// TIA Portal V15.1 export
// export: Created 2020-06-12T07:35:47.2880859Z, ExportSetting None, DisplayName Totally Integrated Automation Portal, DisplayVersion V15.1, DisplayName TIA Portal Openness, DisplayVersion V15.1, DisplayName STEP 7 Professional, DisplayVersion V15.1, DisplayName STEP 7 Safety, DisplayVersion V15.1, DisplayName WinCC Advanced, DisplayVersion V15.1
FUNCTION "Gas_ctrl" : Void   // FC2, FBD
TITLE = Gas system
{ S7_Optimized_Access := 'TRUE' }
// This is a simple 1-line systsem which works in the modes:
// * Keep constant pressure (use fixed flow to reach a target pressure)
// * Keep constant flow (use controllable flow to compensate a gas leakages and a dedusting suction)
// * flood the mold and hood by defined gas volume
// stored: SetENOAutomatically False
   VAR_TEMP
      tActFlow : Real;
      tFloodAmount : Real;   // Temp calculation flood gas amount
      tLinePress : Real;
      tSetFlow : Real;
      tActPress : Real;
      _csf : Bool;
      tRun : Bool;   // Pre Flooding active
      tRunForFlooding : Bool;   // Flooding active
      tDoAmount : Bool;
      tStop : Bool;
      tAutoOn : Bool;
      tReqOn : Bool;
      tReqOff : Bool;
      tReqPressOn : Bool;
      tReqPressOff : Bool;
      tReqAmountOn : Bool;
      tReqAmountOff : Bool;
      tAutoOff : Bool;
      tReqAmountReset : Bool;
      tReqDummy : Bool;
      tGasOn : Bool;
      tAutoMode : Int;
      tMeasFlow : Real;
      tDoPressConst : Bool;
      tDoFlowConst : Bool;
      tCurrSetFlow : Real;
      tAutoIsOn : Bool;
      tPressAboveSet : Real;
      tGasBlowOn : Bool;
   END_VAR
   VAR_TEMP   // added for the SCL form of the ladder/FBD networks
      _w1 : Bool;
      _w2 : Bool;
   END_VAR
BEGIN

REGION Network 1: COMMON SYSTEM FAULT
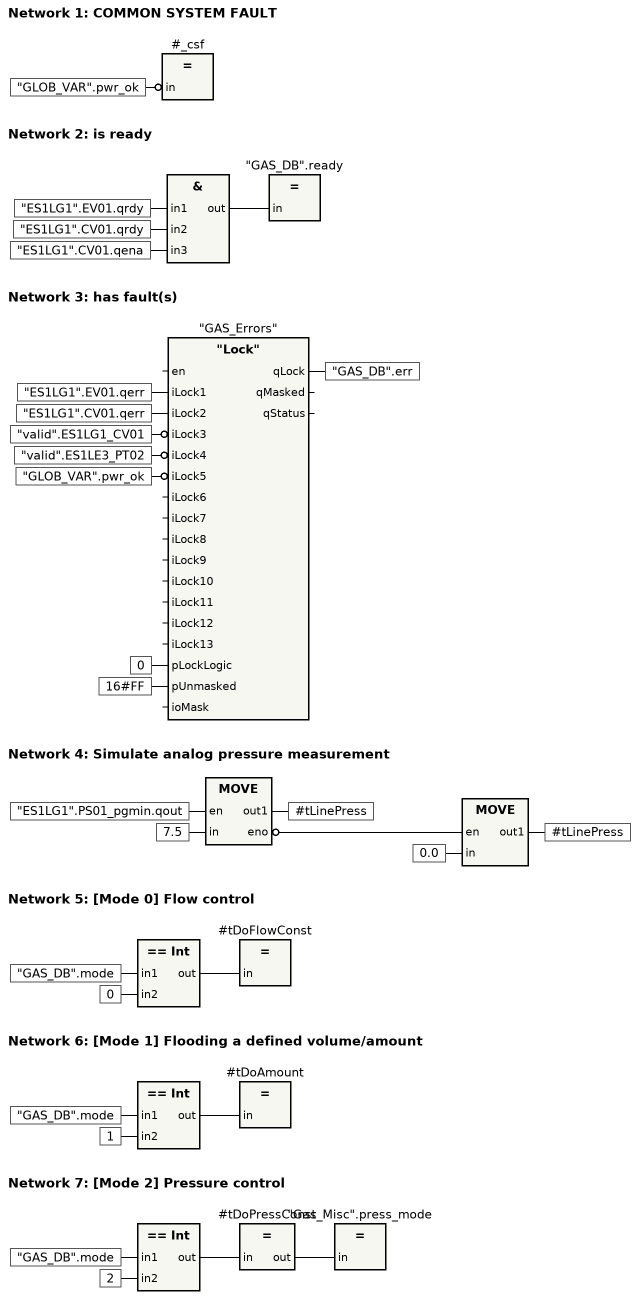
   #_csf := NOT "GLOB_VAR".pwr_ok;
END_REGION

REGION Network 2: is ready
   "GAS_DB".ready := "ES1LG1".EV01.qrdy AND "ES1LG1".CV01.qrdy AND "ES1LG1".CV01.qena;
END_REGION

REGION Network 3: has fault(s)
   "GAS_Errors"(iLock1 := "ES1LG1".EV01.qerr,   // "Lock"
                iLock2 := "ES1LG1".CV01.qerr,
                iLock3 := NOT "valid".ES1LG1_CV01,
                iLock4 := NOT "valid".ES1LE3_PT02,
                iLock5 := NOT "GLOB_VAR".pwr_ok,
                pLockLogic := 0,
                pUnmasked := 16#FF,
                qLock => "GAS_DB".err);
END_REGION

REGION Network 4: Simulate analog pressure measurement
   IF "ES1LG1".PS01_pgmin.qout THEN #tLinePress := 7.5; END_IF;
   IF NOT "ES1LG1".PS01_pgmin.qout THEN #tLinePress := 0.0; END_IF;
END_REGION

REGION Network 5: [Mode 0] Flow control
   #tDoFlowConst := "GAS_DB".mode = 0;
END_REGION

REGION Network 6: [Mode 1] Flooding a defined volume/amount
   #tDoAmount := "GAS_DB".mode = 1;
END_REGION

REGION Network 7: [Mode 2] Pressure control
   #tDoPressConst := "GAS_DB".mode = 2;
   "Gas_Misc".press_mode := #tDoPressConst;
END_REGION

REGION Network 8: Flow set: flow const
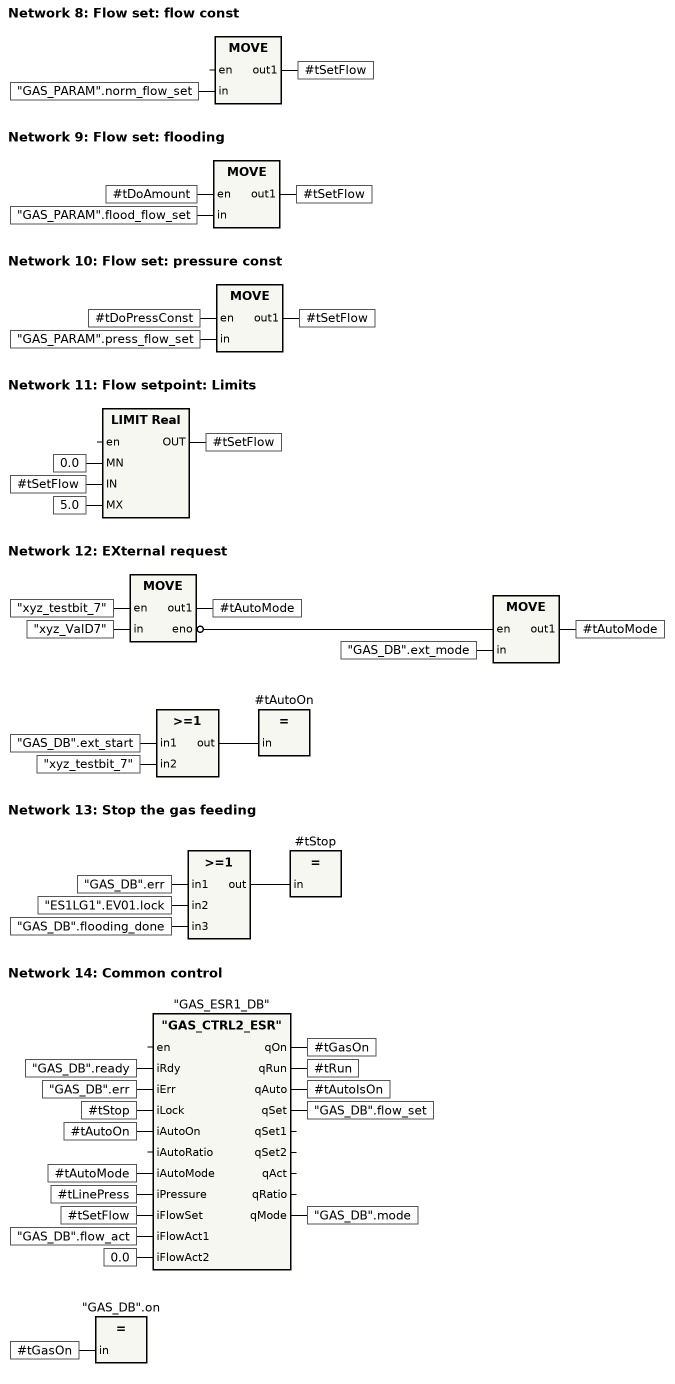
   #tSetFlow := "GAS_PARAM".norm_flow_set;
END_REGION

REGION Network 9: Flow set: flooding
   IF #tDoAmount THEN #tSetFlow := "GAS_PARAM".flood_flow_set; END_IF;
END_REGION

REGION Network 10: Flow set: pressure const
   IF #tDoPressConst THEN #tSetFlow := "GAS_PARAM".press_flow_set; END_IF;
END_REGION

REGION Network 11: Flow setpoint: Limits
   #tSetFlow := LIMIT(MN := 0.0, IN := #tSetFlow, MX := 5.0);
END_REGION

REGION Network 12: EXternal request
   IF "xyz_testbit_7" THEN #tAutoMode := "xyz_ValD7"; END_IF;
   IF NOT "xyz_testbit_7" THEN #tAutoMode := "GAS_DB".ext_mode; END_IF;
   #tAutoOn := "GAS_DB".ext_start OR "xyz_testbit_7";
END_REGION

REGION Network 13: Stop the gas feeding
   #tStop := "GAS_DB".err OR "ES1LG1".EV01.lock OR "GAS_DB".flooding_done;
END_REGION

REGION Network 14: Common control
   "GAS_ESR1_DB"(iRdy := "GAS_DB".ready,   // "GAS_CTRL2_ESR"
                 iErr := "GAS_DB".err,
                 iLock := #tStop,
                 iAutoOn := #tAutoOn,
                 iAutoMode := #tAutoMode,
                 iPressure := #tLinePress,
                 iFlowSet := #tSetFlow,
                 iFlowAct1 := "GAS_DB".flow_act,
                 iFlowAct2 := 0.0,
                 qOn => #tGasOn,
                 qRun => #tRun,
                 qAuto => #tAutoIsOn,
                 qSet => "GAS_DB".flow_set,
                 qMode => "GAS_DB".mode);
   "GAS_DB".on := #tGasOn;
END_REGION

REGION Network 15: M1> Flooding is requested
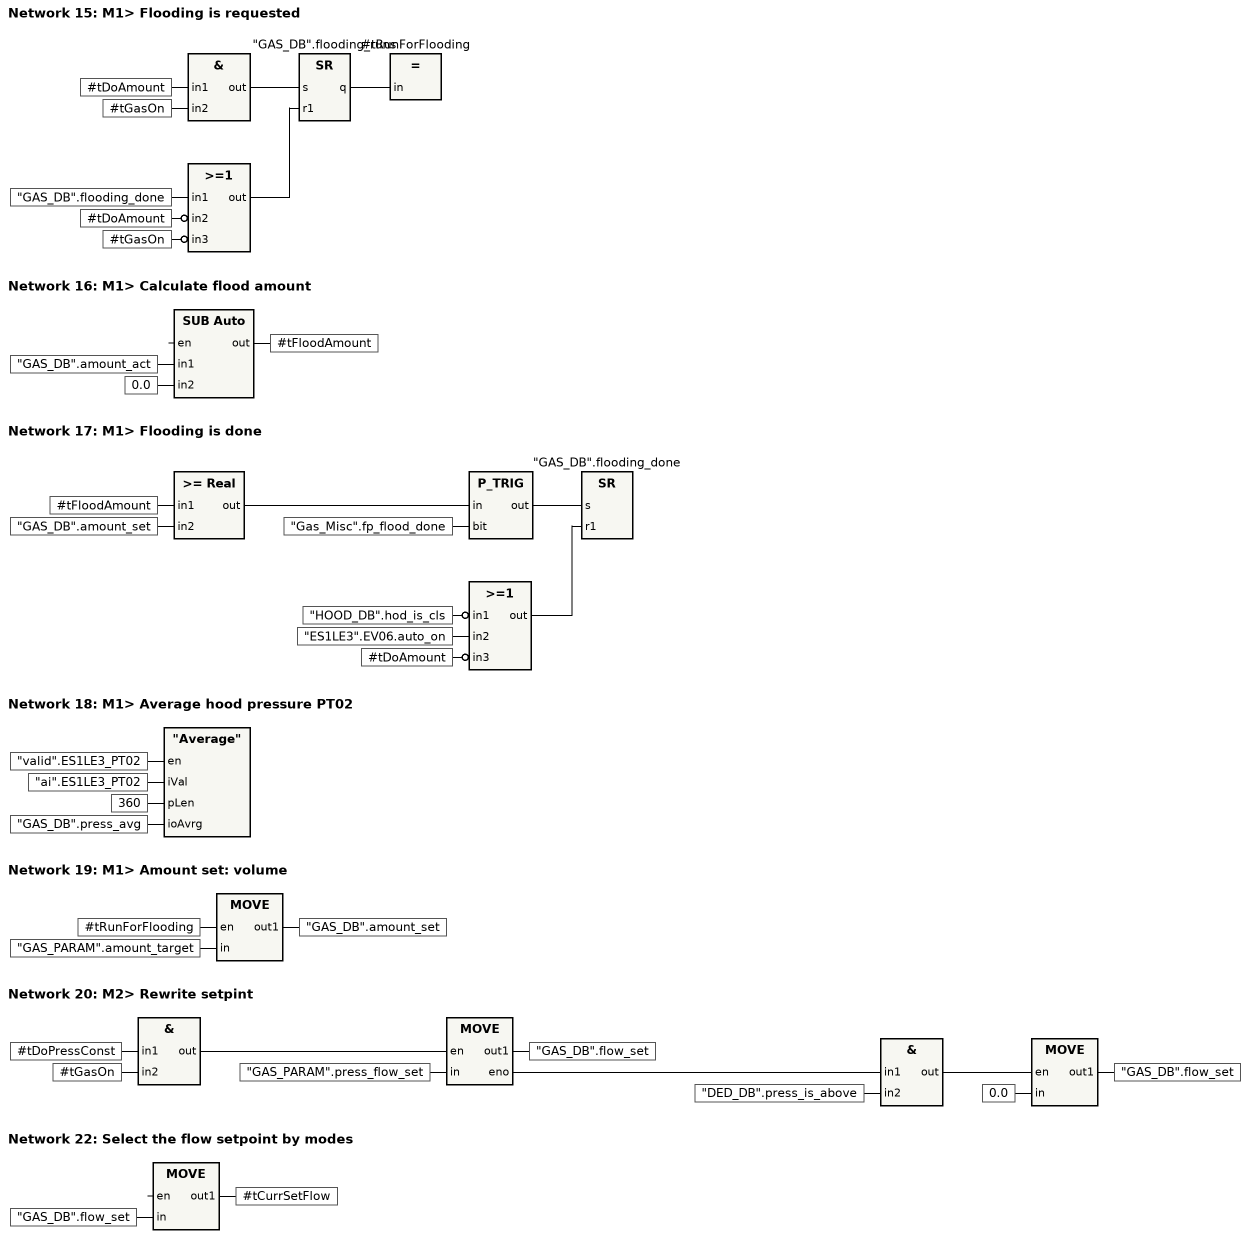
   IF #tDoAmount AND #tGasOn THEN
       "GAS_DB".flooding_runs := TRUE;   // SR flip-flop
   END_IF;
   IF "GAS_DB".flooding_done OR NOT #tDoAmount OR NOT #tGasOn THEN "GAS_DB".flooding_runs := FALSE; END_IF;
   #tRunForFlooding := "GAS_DB".flooding_runs;
END_REGION

REGION Network 16: M1> Calculate flood amount
   #tFloodAmount := "GAS_DB".amount_act - 0.0;
END_REGION

REGION Network 17: M1> Flooding is done
   #_w1 := #tFloodAmount >= "GAS_DB".amount_set;
   #_w2 := #_w1 AND NOT "Gas_Misc".fp_flood_done;   // rising edge
   "Gas_Misc".fp_flood_done := #_w1;
   IF #_w2 THEN
       "GAS_DB".flooding_done := TRUE;   // SR flip-flop
   END_IF;
   IF NOT "HOOD_DB".hod_is_cls OR "ES1LE3".EV06.auto_on OR NOT #tDoAmount THEN
       "GAS_DB".flooding_done := FALSE;
   END_IF;
END_REGION

REGION Network 18: M1> Average hood pressure PT02
   IF "valid".ES1LE3_PT02 THEN
       "Average"(iVal := "ai".ES1LE3_PT02, pLen := 360, ioAvrg := "GAS_DB".press_avg);
   END_IF;
END_REGION

REGION Network 19: M1> Amount set: volume
   IF #tRunForFlooding THEN "GAS_DB".amount_set := "GAS_PARAM".amount_target; END_IF;
END_REGION

REGION Network 20: M2> Rewrite setpint
   // FIXME: this is trick :( It should be re-factored
   #_w1 := #tDoPressConst AND #tGasOn;
   IF #_w1 THEN "GAS_DB".flow_set := "GAS_PARAM".press_flow_set; END_IF;
   IF #_w1 AND "DED_DB".press_is_above THEN "GAS_DB".flow_set := 0.0; END_IF;
END_REGION

REGION Network 21: ******************************
END_REGION

REGION Network 22: Select the flow setpoint by modes
   #tCurrSetFlow := "GAS_DB".flow_set;
END_REGION

REGION Network 23: Actual flow (emulation)
   // THis is using because a measurement is not correct
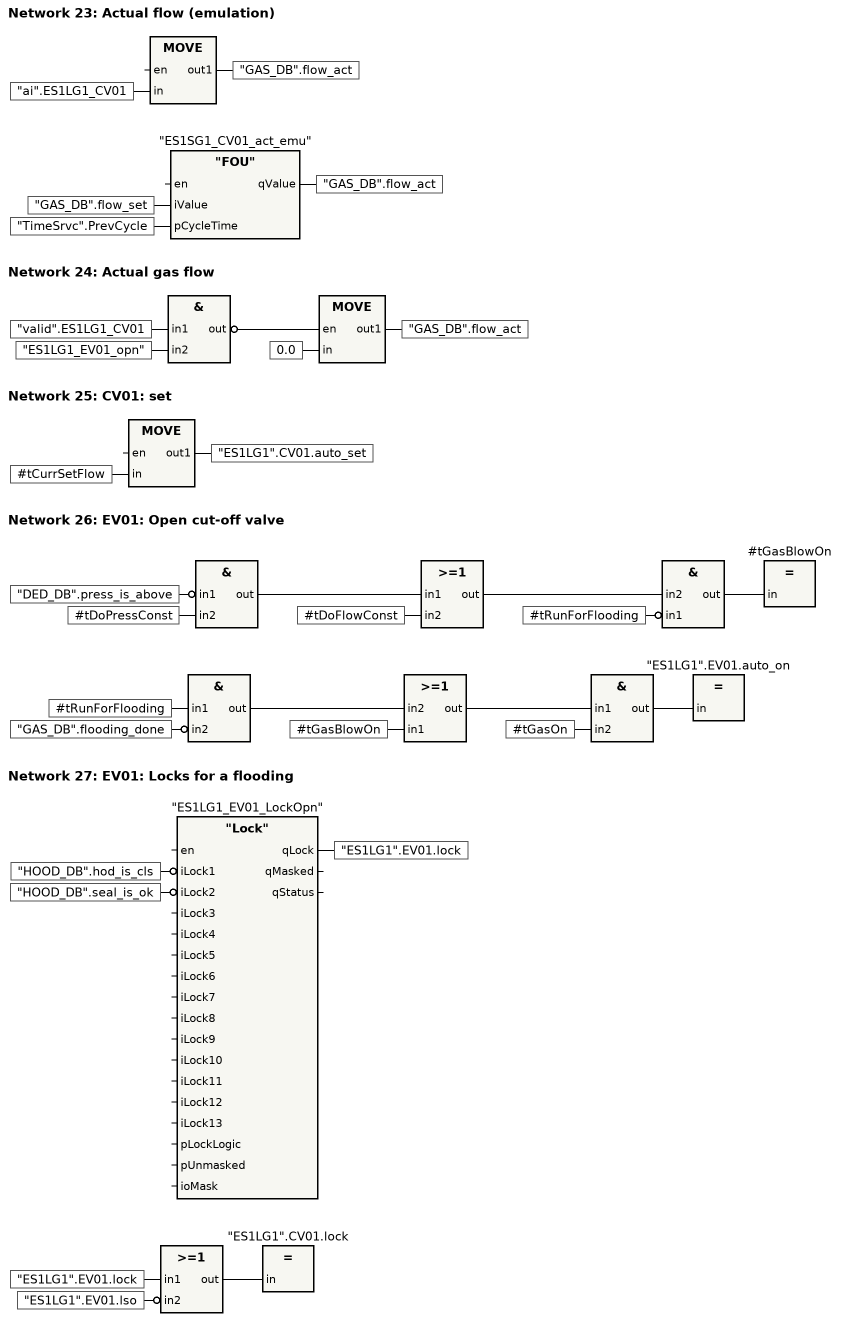
   "GAS_DB".flow_act := "ai".ES1LG1_CV01;
   "ES1SG1_CV01_act_emu"(iValue := "GAS_DB".flow_set,   // "FOU"
                         pCycleTime := "TimeSrvc".PrevCycle,
                         qValue => "GAS_DB".flow_act);
END_REGION

REGION Network 24: Actual gas flow
   IF NOT ("valid".ES1LG1_CV01 AND "ES1LG1_EV01_opn") THEN "GAS_DB".flow_act := 0.0; END_IF;
END_REGION

REGION Network 25: CV01: set
   "ES1LG1".CV01.auto_set := #tCurrSetFlow;
END_REGION

REGION Network 26: EV01: Open cut-off valve
   #tGasBlowOn := ((NOT "DED_DB".press_is_above AND #tDoPressConst) OR #tDoFlowConst) AND NOT #tRunForFlooding;
   "ES1LG1".EV01.auto_on := ((#tRunForFlooding AND NOT "GAS_DB".flooding_done) OR #tGasBlowOn) AND #tGasOn;
END_REGION

REGION Network 27: EV01: Locks for a flooding
   "ES1LG1_EV01_LockOpn"(iLock1 := NOT "HOOD_DB".hod_is_cls,   // "Lock"
                         iLock2 := NOT "HOOD_DB".seal_is_ok,
                         qLock => "ES1LG1".EV01.lock);
   "ES1LG1".CV01.lock := "ES1LG1".EV01.lock OR NOT "ES1LG1".EV01.lso;
END_REGION

REGION Network 28: ******************************
END_REGION

REGION Network 29: Calculate Gas total amount [m3]
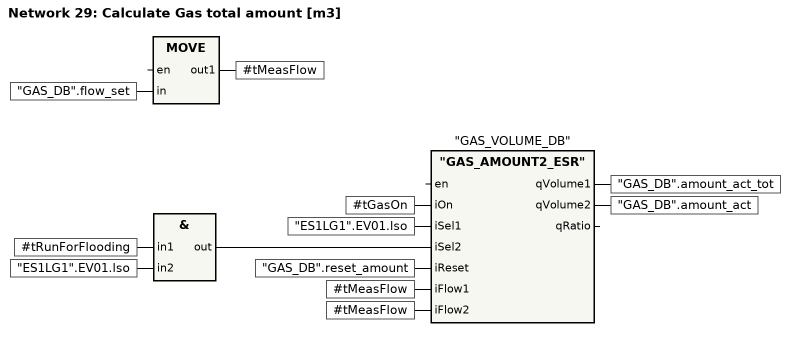
   #tMeasFlow := "GAS_DB".flow_set;
   "GAS_VOLUME_DB"(iOn := #tGasOn,   // "GAS_AMOUNT2_ESR"
                   iSel1 := "ES1LG1".EV01.lso,
                   iSel2 := #tRunForFlooding AND "ES1LG1".EV01.lso,
                   iReset := "GAS_DB".reset_amount,
                   iFlow1 := #tMeasFlow,
                   iFlow2 := #tMeasFlow,
                   qVolume1 => "GAS_DB".amount_act_tot,
                   qVolume2 => "GAS_DB".amount_act);
END_REGION

REGION Network 30: ******************************
END_REGION
END_FUNCTION
